Staubli VAL3: StopAll.pgx

public program StopAll()
  local num l_ni
begin
  for l_ni=0 to nAxesSum-1
    call stopExtAxis(l_ni)
  endFor
end
